RoboDK station: simulation.rdk

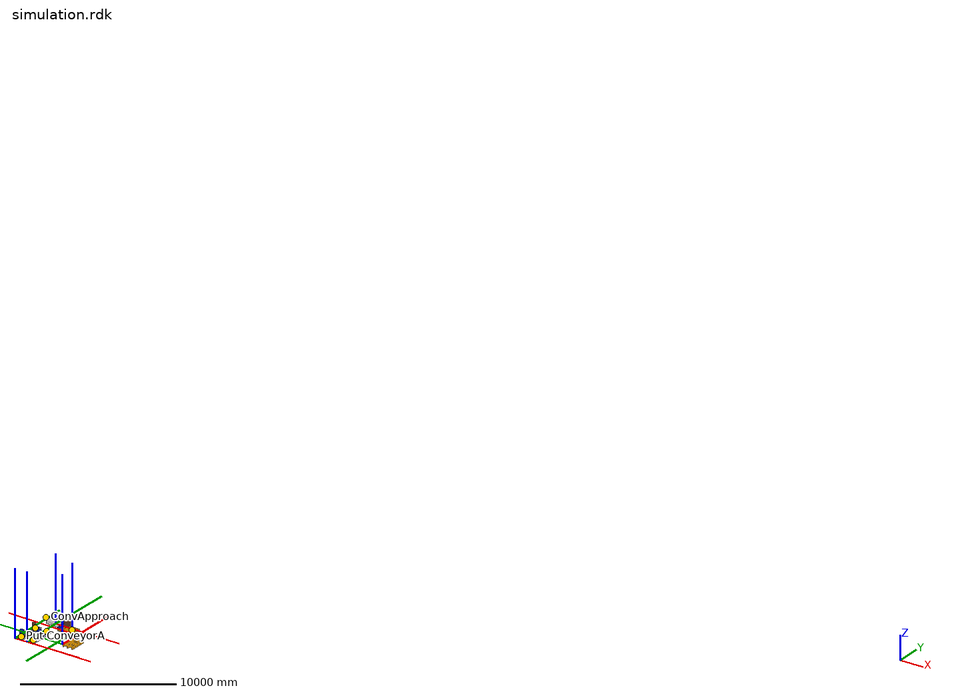
[picture v0: the station drawn from its stored meshes, robots at their saved joint values, targets as dots, program paths as lines]
Station Conveyor simulation. Poses are relative to the parent item; angles as X-Y-Z fixed-axis rotations.
Station parameters (name, value as stored): SizeBox, 150, 300, 150, SizePallet, 3,2,3, ConvSpeed, 40.0, SENSOR, 0, SENSOR-1, 0, SENSOR-2, 0, ROBOT_SWITCHER, 0, TRIGGER-2, 0, TRIGGER-1, 0, SizeBoxA, 240.0,200.0,500.0, SizePalletA, 3,3,3, SizeBoxB, 220.0,190.0,450.0, SizePalletB, 3,3,3, BoxType, 2
  - object box100mm at (0, 0, 0) mm, size 100 x 100 x 100 mm, geometry from box.sld
  - frame ABB IRB 460 Base at (1386.49, 2720.82, 0) mm, rotated rx 0 ry 0 rz -1.04 deg
    - robot ABB IRB 460: 4 axes, payload 110 kg, reach 2400 mm, repeatability 0.2 mm, weight 925 kg
        joint limits [-165, -40, -20, -300] to [165, 85, 120, 300]; home [0, 0, 0, 0]; saved at [-93.5, -29.324, 4.864, 86.5]
      - tool Gripper, TCP at (24.96, -1.82, 200) mm, size 240 x 288 x 203 mm
    - target ConvApproach (joint target) at (-38.73, -1039.73, 855.5) mm, rotated rx -180 ry 0 rz 0 deg; joints [-93.5, -29.324, 4.864, 86.5, 0, 0] of ABB IRB 460
    - target PalletApproach (joint target) at (1357.36, -110.16, 3.72) mm, rotated rx -180 ry 0 rz 0 deg; joints [-4.804, 23.379, 62.26, 175.196, 0, 0] of ABB IRB 460
    - frame PalletB at (545.23, 1038.18, -930) mm, rotated rx 0 ry 0 rz -180 deg
      - object PalletExtension at (1200, -800, 0) mm, rotated rx 0 ry 0 rz 90 deg, size 800 x 144 x 1200 mm, geometry from User Library-Europallet.igs
    - frame Pallet at (973.14, -611.03, -930) mm, rotated rx 0 ry 0 rz 90 deg
      - object Europallet at (1200, -800, 0) mm, rotated rx 0 ry 0 rz 90 deg, size 800 x 144 x 1200 mm, geometry from User Library-Europallet.igs
      - object Part 2 1030.0 685.0 225.0 1.0 at (2351.1, 1457.91, 225) mm, rotated rx -180 ry 0 rz -90 deg, size 220 x 190 x 450 mm, geometry from box.sld
      - object Part 2 1030.0 495.0 225.0 1.0 at (2149.1, 1457.91, 225) mm, rotated rx -180 ry 0 rz -90 deg, size 220 x 190 x 450 mm, geometry from box.sld
      - object Part 1 1080.0 300.0 250.0 1.0 at (1950.1, 1507.91, 250) mm, rotated rx -180 ry 0 rz -90 deg, size 240 x 200 x 500 mm, geometry from box.sld
      - object Part 1 1080.0 100.0 250.0 1.0 at (1779.1, 1507.91, 250) mm, rotated rx -180 ry 0 rz -90 deg, size 240 x 200 x 500 mm, geometry from box.sld
      - object Part 2 810.0 685.0 225.0 1.0 at (2343.1, 1237.91, 225) mm, rotated rx -180 ry 0 rz -90 deg, size 220 x 190 x 450 mm, geometry from box.sld
      - object Part 2 810.0 495.0 225.0 1.0 at (2144.1, 1237.91, 225) mm, rotated rx -180 ry 0 rz -90 deg, size 220 x 190 x 450 mm, geometry from box.sld
  - frame ConveyorReferenceA at (597.23, -679.82, 119.18) mm
    - robot Conveyor BeltA: 1 axes
        modified DH rows (alpha deg, a mm, theta deg, d mm): 0, 0, 0, 0 linear
        base shift (440, 200, 0) mm, rotated rx 0 ry 90 rz 90 deg
        joint limits [-500000] to [500000]; home [0]; saved at [-494037]
      - frame MovingRefA at (0, 0, 0) mm
        - object Part 2 590.0 685.0 225.0 1.0 at (495646.12, 240, 225) mm, rotated rx -180 ry 0 rz 90 deg, size 220 x 190 x 450 mm, geometry from box.sld
        - object Part 1 840.0 100.0 250.0 1.0 at (494259.12, 240, 250) mm, rotated rx -180 ry 0 rz 90 deg, size 240 x 200 x 500 mm, geometry from box.sld
        - object Part 2 590.0 495.0 225.0 1.0 at (494259.12, 240, 225) mm, rotated rx -180 ry 0 rz 90 deg, size 220 x 190 x 450 mm, geometry from box.sld
        - object Part 1 600.0 300.0 250.0 1.0 at (494259.12, 240, 250) mm, rotated rx -180 ry 0 rz 90 deg, size 240 x 200 x 500 mm, geometry from box.sld
        - object Part 1 600.0 100.0 250.0 1.0 at (494259.12, 240, 250) mm, rotated rx -180 ry 0 rz 90 deg, size 240 x 200 x 500 mm, geometry from box.sld
        - object Part 2 370.0 305.0 225.0 1.0 at (494259.12, 240, 225) mm, rotated rx -180 ry 0 rz 90 deg, size 220 x 190 x 450 mm, geometry from box.sld
        - object Part 2 150.0 305.0 225.0 1.0 at (494259.12, 240, 225) mm, rotated rx -180 ry 0 rz 90 deg, size 220 x 190 x 450 mm, geometry from box.sld
        - object Part 2 1030.0 685.0 675.0 2.0 at (494259.12, 240, 225) mm, rotated rx -180 ry 0 rz 90 deg, size 220 x 190 x 450 mm, geometry from box.sld
        - object Part 1 1080.0 300.0 750.0 2.0 at (494259.12, 240, 250) mm, rotated rx -180 ry 0 rz 90 deg, size 240 x 200 x 500 mm, geometry from box.sld
        - object Part 2 810.0 685.0 675.0 2.0 at (494259.12, 240, 225) mm, rotated rx -180 ry 0 rz 90 deg, size 220 x 190 x 450 mm, geometry from box.sld
        - object Part 2 590.0 685.0 675.0 2.0 at (494259.12, 240, 225) mm, rotated rx -180 ry 0 rz 90 deg, size 220 x 190 x 450 mm, geometry from box.sld
        - object Part 1 840.0 100.0 750.0 2.0 at (494259.12, 240, 250) mm, rotated rx -180 ry 0 rz 90 deg, size 240 x 200 x 500 mm, geometry from box.sld
        - object Part 2 590.0 495.0 675.0 2.0 at (494259.12, 240, 225) mm, rotated rx -180 ry 0 rz 90 deg, size 220 x 190 x 450 mm, geometry from box.sld
        - object Part 1 600.0 300.0 750.0 2.0 at (494259.12, 240, 250) mm, rotated rx -180 ry 0 rz 90 deg, size 240 x 200 x 500 mm, geometry from box.sld
        - object Part 1 600.0 100.0 750.0 2.0 at (494259.12, 240, 250) mm, rotated rx -180 ry 0 rz 90 deg, size 240 x 200 x 500 mm, geometry from box.sld
        - object Part 2 370.0 305.0 675.0 2.0 at (494259.12, 240, 225) mm, rotated rx -180 ry 0 rz 90 deg, size 220 x 190 x 450 mm, geometry from box.sld
        - object Part 2 150.0 305.0 675.0 2.0 at (494259.12, 240, 225) mm, rotated rx -180 ry 0 rz 90 deg, size 220 x 190 x 450 mm, geometry from box.sld
        - object Part 2 1030.0 685.0 1125.0 3.0 at (494259.12, 240, 225) mm, rotated rx -180 ry 0 rz 90 deg, size 220 x 190 x 450 mm, geometry from box.sld
        - object Part 1 1080.0 300.0 1250.0 3.0 at (494259.12, 240, 250) mm, rotated rx -180 ry 0 rz 90 deg, size 240 x 200 x 500 mm, geometry from box.sld
        - object Part 2 810.0 685.0 1125.0 3.0 at (494259.12, 240, 225) mm, rotated rx -180 ry 0 rz 90 deg, size 220 x 190 x 450 mm, geometry from box.sld
        - object Part 2 590.0 685.0 1125.0 3.0 at (494259.12, 240, 225) mm, rotated rx -180 ry 0 rz 90 deg, size 220 x 190 x 450 mm, geometry from box.sld
        - object Part 1 840.0 100.0 1250.0 3.0 at (494259.12, 240, 250) mm, rotated rx -180 ry 0 rz 90 deg, size 240 x 200 x 500 mm, geometry from box.sld
        - object Part 2 590.0 495.0 1125.0 3.0 at (494259.12, 240, 225) mm, rotated rx -180 ry 0 rz 90 deg, size 220 x 190 x 450 mm, geometry from box.sld
        - object Part 1 600.0 300.0 1250.0 3.0 at (494259.12, 240, 250) mm, rotated rx -180 ry 0 rz 90 deg, size 240 x 200 x 500 mm, geometry from box.sld
        - object Part 1 600.0 100.0 1250.0 3.0 at (494259.12, 240, 250) mm, rotated rx -180 ry 0 rz 90 deg, size 240 x 200 x 500 mm, geometry from box.sld
        - object Part 2 370.0 305.0 1125.0 3.0 at (494259.12, 240, 225) mm, rotated rx -180 ry 0 rz 90 deg, size 220 x 190 x 450 mm, geometry from box.sld
        - object Part 2 150.0 305.0 1125.0 3.0 at (494259.12, 240, 225) mm, rotated rx -180 ry 0 rz 90 deg, size 220 x 190 x 450 mm, geometry from box.sld
        - object Part 2 1030.0 685.0 1575.0 4.0 at (494259.12, 240, 225) mm, rotated rx -180 ry 0 rz 90 deg, size 220 x 190 x 450 mm, geometry from box.sld
        - object Part 1 1080.0 300.0 1750.0 4.0 at (494259.12, 240, 250) mm, rotated rx -180 ry 0 rz 90 deg, size 240 x 200 x 500 mm, geometry from box.sld
        - object Part 2 810.0 685.0 1575.0 4.0 at (494259.12, 240, 225) mm, rotated rx -180 ry 0 rz 90 deg, size 220 x 190 x 450 mm, geometry from box.sld
        - object Part 2 590.0 685.0 1575.0 4.0 at (494259.12, 240, 225) mm, rotated rx -180 ry 0 rz 90 deg, size 220 x 190 x 450 mm, geometry from box.sld
        - object Part 1 840.0 100.0 1750.0 4.0 at (494259.12, 240, 250) mm, rotated rx -180 ry 0 rz 90 deg, size 240 x 200 x 500 mm, geometry from box.sld
        - object Part 2 590.0 495.0 1575.0 4.0 at (494259.12, 240, 225) mm, rotated rx -180 ry 0 rz 90 deg, size 220 x 190 x 450 mm, geometry from box.sld
        - object Part 1 600.0 300.0 1750.0 4.0 at (494259.12, 240, 250) mm, rotated rx -180 ry 0 rz 90 deg, size 240 x 200 x 500 mm, geometry from box.sld
        - object Part 1 600.0 100.0 1750.0 4.0 at (494259.12, 240, 250) mm, rotated rx -180 ry 0 rz 90 deg, size 240 x 200 x 500 mm, geometry from box.sld
        - object Part 2 370.0 305.0 1575.0 4.0 at (494259.12, 240, 225) mm, rotated rx -180 ry 0 rz 90 deg, size 220 x 190 x 450 mm, geometry from box.sld
        - object Part 2 150.0 305.0 1575.0 4.0 at (494259.12, 240, 225) mm, rotated rx -180 ry 0 rz 90 deg, size 220 x 190 x 450 mm, geometry from box.sld
        - object Part 2 1030.0 685.0 225.0 1.0 at (494259.12, 240, 225) mm, rotated rx -180 ry 0 rz 90 deg, size 220 x 190 x 450 mm, geometry from box.sld
        - object Part 1 1080.0 300.0 250.0 1.0 at (494259.12, 240, 250) mm, rotated rx -180 ry 0 rz 90 deg, size 240 x 200 x 500 mm, geometry from box.sld
        - object Part 2 810.0 685.0 225.0 1.0 at (494259.12, 240, 225) mm, rotated rx -180 ry 0 rz 90 deg, size 220 x 190 x 450 mm, geometry from box.sld
        - object Part 2 590.0 685.0 225.0 1.0 at (494259.12, 240, 225) mm, rotated rx -180 ry 0 rz 90 deg, size 220 x 190 x 450 mm, geometry from box.sld
        - object Part 1 840.0 100.0 250.0 1.0 at (494259.12, 240, 250) mm, rotated rx -180 ry 0 rz 90 deg, size 240 x 200 x 500 mm, geometry from box.sld
        - object Part 2 590.0 495.0 225.0 1.0 at (494259.12, 240, 225) mm, rotated rx -180 ry 0 rz 90 deg, size 220 x 190 x 450 mm, geometry from box.sld
        - object Part 1 600.0 300.0 250.0 1.0 at (494259.12, 240, 250) mm, rotated rx -180 ry 0 rz 90 deg, size 240 x 200 x 500 mm, geometry from box.sld
        - object Part 1 600.0 100.0 250.0 1.0 at (494259.12, 240, 250) mm, rotated rx -180 ry 0 rz 90 deg, size 240 x 200 x 500 mm, geometry from box.sld
        - object Part 2 370.0 305.0 225.0 1.0 at (494259.12, 240, 225) mm, rotated rx -180 ry 0 rz 90 deg, size 220 x 190 x 450 mm, geometry from box.sld
        - object Part 2 150.0 305.0 225.0 1.0 at (494259.12, 240, 225) mm, rotated rx -180 ry 0 rz 90 deg, size 220 x 190 x 450 mm, geometry from box.sld
        - object Part 2 1030.0 685.0 675.0 2.0 at (494259.12, 240, 225) mm, rotated rx -180 ry 0 rz 90 deg, size 220 x 190 x 450 mm, geometry from box.sld
        - object Part 1 1080.0 300.0 750.0 2.0 at (494259.12, 240, 250) mm, rotated rx -180 ry 0 rz 90 deg, size 240 x 200 x 500 mm, geometry from box.sld
        - object Part 2 810.0 685.0 675.0 2.0 at (494259.12, 240, 225) mm, rotated rx -180 ry 0 rz 90 deg, size 220 x 190 x 450 mm, geometry from box.sld
        - object Part 2 590.0 685.0 675.0 2.0 at (494259.12, 240, 225) mm, rotated rx -180 ry 0 rz 90 deg, size 220 x 190 x 450 mm, geometry from box.sld
        - object Part 1 840.0 100.0 750.0 2.0 at (494259.12, 240, 250) mm, rotated rx -180 ry 0 rz 90 deg, size 240 x 200 x 500 mm, geometry from box.sld
        - object Part 2 590.0 495.0 675.0 2.0 at (494259.12, 240, 225) mm, rotated rx -180 ry 0 rz 90 deg, size 220 x 190 x 450 mm, geometry from box.sld
        - object Part 1 600.0 300.0 750.0 2.0 at (494259.12, 240, 250) mm, rotated rx -180 ry 0 rz 90 deg, size 240 x 200 x 500 mm, geometry from box.sld
        - object Part 1 600.0 100.0 750.0 2.0 at (494259.12, 240, 250) mm, rotated rx -180 ry 0 rz 90 deg, size 240 x 200 x 500 mm, geometry from box.sld
        - object Part 2 370.0 305.0 675.0 2.0 at (494259.12, 240, 225) mm, rotated rx -180 ry 0 rz 90 deg, size 220 x 190 x 450 mm, geometry from box.sld
        - object Part 2 150.0 305.0 675.0 2.0 at (494259.12, 240, 225) mm, rotated rx -180 ry 0 rz 90 deg, size 220 x 190 x 450 mm, geometry from box.sld
        - object Part 2 1030.0 685.0 1125.0 3.0 at (494259.12, 240, 225) mm, rotated rx -180 ry 0 rz 90 deg, size 220 x 190 x 450 mm, geometry from box.sld
        - object Part 1 1080.0 300.0 1250.0 3.0 at (494259.12, 240, 250) mm, rotated rx -180 ry 0 rz 90 deg, size 240 x 200 x 500 mm, geometry from box.sld
        - object Part 2 810.0 685.0 1125.0 3.0 at (494259.12, 240, 225) mm, rotated rx -180 ry 0 rz 90 deg, size 220 x 190 x 450 mm, geometry from box.sld
        - object Part 2 590.0 685.0 1125.0 3.0 at (494259.12, 240, 225) mm, rotated rx -180 ry 0 rz 90 deg, size 220 x 190 x 450 mm, geometry from box.sld
        - object Part 1 840.0 100.0 1250.0 3.0 at (494259.12, 240, 250) mm, rotated rx -180 ry 0 rz 90 deg, size 240 x 200 x 500 mm, geometry from box.sld
        - object Part 2 590.0 495.0 1125.0 3.0 at (494259.12, 240, 225) mm, rotated rx -180 ry 0 rz 90 deg, size 220 x 190 x 450 mm, geometry from box.sld
        - object Part 1 600.0 300.0 1250.0 3.0 at (494259.12, 240, 250) mm, rotated rx -180 ry 0 rz 90 deg, size 240 x 200 x 500 mm, geometry from box.sld
        - object Part 1 600.0 100.0 1250.0 3.0 at (494259.12, 240, 250) mm, rotated rx -180 ry 0 rz 90 deg, size 240 x 200 x 500 mm, geometry from box.sld
        - object Part 2 370.0 305.0 1125.0 3.0 at (494259.12, 240, 225) mm, rotated rx -180 ry 0 rz 90 deg, size 220 x 190 x 450 mm, geometry from box.sld
        - object Part 2 150.0 305.0 1125.0 3.0 at (494259.12, 240, 225) mm, rotated rx -180 ry 0 rz 90 deg, size 220 x 190 x 450 mm, geometry from box.sld
        - object Part 2 1030.0 685.0 1575.0 4.0 at (494259.12, 240, 225) mm, rotated rx -180 ry 0 rz 90 deg, size 220 x 190 x 450 mm, geometry from box.sld
        - object Part 1 1080.0 300.0 1750.0 4.0 at (494259.12, 240, 250) mm, rotated rx -180 ry 0 rz 90 deg, size 240 x 200 x 500 mm, geometry from box.sld
        - object Part 2 810.0 685.0 1575.0 4.0 at (494259.12, 240, 225) mm, rotated rx -180 ry 0 rz 90 deg, size 220 x 190 x 450 mm, geometry from box.sld
        - object Part 2 590.0 685.0 1575.0 4.0 at (494259.12, 240, 225) mm, rotated rx -180 ry 0 rz 90 deg, size 220 x 190 x 450 mm, geometry from box.sld
        - object Part 1 840.0 100.0 1750.0 4.0 at (494259.12, 240, 250) mm, rotated rx -180 ry 0 rz 90 deg, size 240 x 200 x 500 mm, geometry from box.sld
        - object Part 2 590.0 495.0 1575.0 4.0 at (494259.12, 240, 225) mm, rotated rx -180 ry 0 rz 90 deg, size 220 x 190 x 450 mm, geometry from box.sld
        - object Part 1 600.0 300.0 1750.0 4.0 at (494259.12, 240, 250) mm, rotated rx -180 ry 0 rz 90 deg, size 240 x 200 x 500 mm, geometry from box.sld
        - object Part 1 600.0 100.0 1750.0 4.0 at (494259.12, 240, 250) mm, rotated rx -180 ry 0 rz 90 deg, size 240 x 200 x 500 mm, geometry from box.sld
        - object Part 2 370.0 305.0 1575.0 4.0 at (494259.12, 240, 225) mm, rotated rx -180 ry 0 rz 90 deg, size 220 x 190 x 450 mm, geometry from box.sld
        - object Part 2 150.0 305.0 1575.0 4.0 at (494259.12, 240, 225) mm, rotated rx -180 ry 0 rz 90 deg, size 220 x 190 x 450 mm, geometry from box.sld
    - target ConveyorHomeA (joint target) at (440, 200, 0) mm, rotated rx 0 ry 0 rz 90 deg; joints [0] of Conveyor BeltA
    - target ConveyorMoveA (joint target) at (440, 99999, 0) mm, rotated rx 0 ry 0 rz 90 deg; joints [99799] of Conveyor BeltA
    - object Sensor SICK WL4S-1 at (551, 1930, 24) mm, rotated rx 90 ry 0 rz 180 deg, size 683.3 x 45.2 x 12.5 mm, geometry from SICK WL4S-3P1330-Order no.1042068 (1).stp
    - target Get ConveyorA (Cartesian target) at (200, 1950, 0) mm, rotated rx -180 ry 0 rz 0 deg; joints [-111.887, 26.233, 48.865, -292.923, 0, 0] of ABB IRB 460
    - target Put ConveyorA (Cartesian target) at (200, 422.12, 0) mm, rotated rx -180 ry 0 rz 180 deg; joints [164.915, -63.548, 110.129, -136.581, -90, -15.085]
  - frame ConveyorReferenceB at (1500, -679.82, 119.18) mm
    - robot Conveyor BeltB: 1 axes
        modified DH rows (alpha deg, a mm, theta deg, d mm): 0, 0, 0, 0 linear
        base shift (440, 200, 0) mm, rotated rx 0 ry 90 rz 90 deg
        joint limits [-500000] to [500000]; home [0]; saved at [-494159]
      - frame MovingRefB at (0, 0, 0) mm
        - object Part 1 840.0 300.0 250.0 1.0 at (495052.11, 240, 250) mm, rotated rx -180 ry 0 rz 90 deg, size 240 x 200 x 500 mm, geometry from box.sld
        - object Part 1 360.0 700.0 250.0 1.0 at (494381.11, 240, 250) mm, rotated rx -180 ry 0 rz 90 deg, size 240 x 200 x 500 mm, geometry from box.sld
        - object Part 1 120.0 700.0 250.0 1.0 at (494381.11, 240, 250) mm, rotated rx -180 ry 0 rz 90 deg, size 240 x 200 x 500 mm, geometry from box.sld
        - object Part 1 360.0 500.0 250.0 1.0 at (494381.11, 240, 250) mm, rotated rx -180 ry 0 rz 90 deg, size 240 x 200 x 500 mm, geometry from box.sld
        - object Part 1 120.0 500.0 250.0 1.0 at (494381.11, 240, 250) mm, rotated rx -180 ry 0 rz 90 deg, size 240 x 200 x 500 mm, geometry from box.sld
        - object Part 2 370.0 115.0 225.0 1.0 at (494381.11, 240, 225) mm, rotated rx -180 ry 0 rz 90 deg, size 220 x 190 x 450 mm, geometry from box.sld
        - object Part 2 150.0 115.0 225.0 1.0 at (494381.11, 240, 225) mm, rotated rx -180 ry 0 rz 90 deg, size 220 x 190 x 450 mm, geometry from box.sld
        - object Part 2 1030.0 495.0 675.0 2.0 at (494381.11, 240, 225) mm, rotated rx -180 ry 0 rz 90 deg, size 220 x 190 x 450 mm, geometry from box.sld
        - object Part 1 1080.0 100.0 750.0 2.0 at (494381.11, 240, 250) mm, rotated rx -180 ry 0 rz 90 deg, size 240 x 200 x 500 mm, geometry from box.sld
        - object Part 2 810.0 495.0 675.0 2.0 at (494381.11, 240, 225) mm, rotated rx -180 ry 0 rz 90 deg, size 220 x 190 x 450 mm, geometry from box.sld
        - object Part 1 840.0 300.0 750.0 2.0 at (494381.11, 240, 250) mm, rotated rx -180 ry 0 rz 90 deg, size 240 x 200 x 500 mm, geometry from box.sld
        - object Part 1 360.0 700.0 750.0 2.0 at (494381.11, 240, 250) mm, rotated rx -180 ry 0 rz 90 deg, size 240 x 200 x 500 mm, geometry from box.sld
        - object Part 1 120.0 700.0 750.0 2.0 at (494381.11, 240, 250) mm, rotated rx -180 ry 0 rz 90 deg, size 240 x 200 x 500 mm, geometry from box.sld
        - object Part 1 360.0 500.0 750.0 2.0 at (494381.11, 240, 250) mm, rotated rx -180 ry 0 rz 90 deg, size 240 x 200 x 500 mm, geometry from box.sld
        - object Part 1 120.0 500.0 750.0 2.0 at (494381.11, 240, 250) mm, rotated rx -180 ry 0 rz 90 deg, size 240 x 200 x 500 mm, geometry from box.sld
        - object Part 2 370.0 115.0 675.0 2.0 at (494381.11, 240, 225) mm, rotated rx -180 ry 0 rz 90 deg, size 220 x 190 x 450 mm, geometry from box.sld
        - object Part 2 150.0 115.0 675.0 2.0 at (494381.11, 240, 225) mm, rotated rx -180 ry 0 rz 90 deg, size 220 x 190 x 450 mm, geometry from box.sld
        - object Part 2 1030.0 495.0 1125.0 3.0 at (494381.11, 240, 225) mm, rotated rx -180 ry 0 rz 90 deg, size 220 x 190 x 450 mm, geometry from box.sld
        - object Part 1 1080.0 100.0 1250.0 3.0 at (494381.11, 240, 250) mm, rotated rx -180 ry 0 rz 90 deg, size 240 x 200 x 500 mm, geometry from box.sld
        - object Part 2 810.0 495.0 1125.0 3.0 at (494381.11, 240, 225) mm, rotated rx -180 ry 0 rz 90 deg, size 220 x 190 x 450 mm, geometry from box.sld
        - object Part 1 840.0 300.0 1250.0 3.0 at (494381.11, 240, 250) mm, rotated rx -180 ry 0 rz 90 deg, size 240 x 200 x 500 mm, geometry from box.sld
        - object Part 1 360.0 700.0 1250.0 3.0 at (494381.11, 240, 250) mm, rotated rx -180 ry 0 rz 90 deg, size 240 x 200 x 500 mm, geometry from box.sld
        - object Part 1 120.0 700.0 1250.0 3.0 at (494381.11, 240, 250) mm, rotated rx -180 ry 0 rz 90 deg, size 240 x 200 x 500 mm, geometry from box.sld
        - object Part 1 360.0 500.0 1250.0 3.0 at (494381.11, 240, 250) mm, rotated rx -180 ry 0 rz 90 deg, size 240 x 200 x 500 mm, geometry from box.sld
        - object Part 1 120.0 500.0 1250.0 3.0 at (494381.11, 240, 250) mm, rotated rx -180 ry 0 rz 90 deg, size 240 x 200 x 500 mm, geometry from box.sld
        - object Part 2 370.0 115.0 1125.0 3.0 at (494381.11, 240, 225) mm, rotated rx -180 ry 0 rz 90 deg, size 220 x 190 x 450 mm, geometry from box.sld
        - object Part 2 150.0 115.0 1125.0 3.0 at (494381.11, 240, 225) mm, rotated rx -180 ry 0 rz 90 deg, size 220 x 190 x 450 mm, geometry from box.sld
        - object Part 2 1030.0 495.0 1575.0 4.0 at (494381.11, 240, 225) mm, rotated rx -180 ry 0 rz 90 deg, size 220 x 190 x 450 mm, geometry from box.sld
        - object Part 1 1080.0 100.0 1750.0 4.0 at (494381.11, 240, 250) mm, rotated rx -180 ry 0 rz 90 deg, size 240 x 200 x 500 mm, geometry from box.sld
        - object Part 2 810.0 495.0 1575.0 4.0 at (494381.11, 240, 225) mm, rotated rx -180 ry 0 rz 90 deg, size 220 x 190 x 450 mm, geometry from box.sld
        - object Part 1 840.0 300.0 1750.0 4.0 at (494381.11, 240, 250) mm, rotated rx -180 ry 0 rz 90 deg, size 240 x 200 x 500 mm, geometry from box.sld
        - object Part 1 360.0 700.0 1750.0 4.0 at (494381.11, 240, 250) mm, rotated rx -180 ry 0 rz 90 deg, size 240 x 200 x 500 mm, geometry from box.sld
        - object Part 1 120.0 700.0 1750.0 4.0 at (494381.11, 240, 250) mm, rotated rx -180 ry 0 rz 90 deg, size 240 x 200 x 500 mm, geometry from box.sld
        - object Part 1 360.0 500.0 1750.0 4.0 at (494381.11, 240, 250) mm, rotated rx -180 ry 0 rz 90 deg, size 240 x 200 x 500 mm, geometry from box.sld
        - object Part 1 120.0 500.0 1750.0 4.0 at (494381.11, 240, 250) mm, rotated rx -180 ry 0 rz 90 deg, size 240 x 200 x 500 mm, geometry from box.sld
        - object Part 2 370.0 115.0 1575.0 4.0 at (494381.11, 240, 225) mm, rotated rx -180 ry 0 rz 90 deg, size 220 x 190 x 450 mm, geometry from box.sld
        - object Part 2 150.0 115.0 1575.0 4.0 at (494381.11, 240, 225) mm, rotated rx -180 ry 0 rz 90 deg, size 220 x 190 x 450 mm, geometry from box.sld
        - object Part 2 1030.0 495.0 225.0 1.0 at (494381.11, 240, 225) mm, rotated rx -180 ry 0 rz 90 deg, size 220 x 190 x 450 mm, geometry from box.sld
        - object Part 1 1080.0 100.0 250.0 1.0 at (494381.11, 240, 250) mm, rotated rx -180 ry 0 rz 90 deg, size 240 x 200 x 500 mm, geometry from box.sld
        - object Part 2 810.0 495.0 225.0 1.0 at (494381.11, 240, 225) mm, rotated rx -180 ry 0 rz 90 deg, size 220 x 190 x 450 mm, geometry from box.sld
        - object Part 1 840.0 300.0 250.0 1.0 at (494381.11, 240, 250) mm, rotated rx -180 ry 0 rz 90 deg, size 240 x 200 x 500 mm, geometry from box.sld
        - object Part 1 360.0 700.0 250.0 1.0 at (494381.11, 240, 250) mm, rotated rx -180 ry 0 rz 90 deg, size 240 x 200 x 500 mm, geometry from box.sld
        - object Part 1 120.0 700.0 250.0 1.0 at (494381.11, 240, 250) mm, rotated rx -180 ry 0 rz 90 deg, size 240 x 200 x 500 mm, geometry from box.sld
        - object Part 1 360.0 500.0 250.0 1.0 at (494381.11, 240, 250) mm, rotated rx -180 ry 0 rz 90 deg, size 240 x 200 x 500 mm, geometry from box.sld
        - object Part 1 120.0 500.0 250.0 1.0 at (494381.11, 240, 250) mm, rotated rx -180 ry 0 rz 90 deg, size 240 x 200 x 500 mm, geometry from box.sld
        - object Part 2 370.0 115.0 225.0 1.0 at (494381.11, 240, 225) mm, rotated rx -180 ry 0 rz 90 deg, size 220 x 190 x 450 mm, geometry from box.sld
        - object Part 2 150.0 115.0 225.0 1.0 at (494381.11, 240, 225) mm, rotated rx -180 ry 0 rz 90 deg, size 220 x 190 x 450 mm, geometry from box.sld
        - object Part 2 1030.0 495.0 675.0 2.0 at (494381.11, 240, 225) mm, rotated rx -180 ry 0 rz 90 deg, size 220 x 190 x 450 mm, geometry from box.sld
        - object Part 1 1080.0 100.0 750.0 2.0 at (494381.11, 240, 250) mm, rotated rx -180 ry 0 rz 90 deg, size 240 x 200 x 500 mm, geometry from box.sld
        - object Part 2 810.0 495.0 675.0 2.0 at (494381.11, 240, 225) mm, rotated rx -180 ry 0 rz 90 deg, size 220 x 190 x 450 mm, geometry from box.sld
        - object Part 1 840.0 300.0 750.0 2.0 at (494381.11, 240, 250) mm, rotated rx -180 ry 0 rz 90 deg, size 240 x 200 x 500 mm, geometry from box.sld
        - object Part 1 360.0 700.0 750.0 2.0 at (494381.11, 240, 250) mm, rotated rx -180 ry 0 rz 90 deg, size 240 x 200 x 500 mm, geometry from box.sld
        - object Part 1 120.0 700.0 750.0 2.0 at (494381.11, 240, 250) mm, rotated rx -180 ry 0 rz 90 deg, size 240 x 200 x 500 mm, geometry from box.sld
        - object Part 1 360.0 500.0 750.0 2.0 at (494381.11, 240, 250) mm, rotated rx -180 ry 0 rz 90 deg, size 240 x 200 x 500 mm, geometry from box.sld
        - object Part 1 120.0 500.0 750.0 2.0 at (494381.11, 240, 250) mm, rotated rx -180 ry 0 rz 90 deg, size 240 x 200 x 500 mm, geometry from box.sld
        - object Part 2 370.0 115.0 675.0 2.0 at (494381.11, 240, 225) mm, rotated rx -180 ry 0 rz 90 deg, size 220 x 190 x 450 mm, geometry from box.sld
        - object Part 2 150.0 115.0 675.0 2.0 at (494381.11, 240, 225) mm, rotated rx -180 ry 0 rz 90 deg, size 220 x 190 x 450 mm, geometry from box.sld
        - object Part 2 1030.0 495.0 1125.0 3.0 at (494381.11, 240, 225) mm, rotated rx -180 ry 0 rz 90 deg, size 220 x 190 x 450 mm, geometry from box.sld
        - object Part 1 1080.0 100.0 1250.0 3.0 at (494381.11, 240, 250) mm, rotated rx -180 ry 0 rz 90 deg, size 240 x 200 x 500 mm, geometry from box.sld
        - object Part 2 810.0 495.0 1125.0 3.0 at (494381.11, 240, 225) mm, rotated rx -180 ry 0 rz 90 deg, size 220 x 190 x 450 mm, geometry from box.sld
        - object Part 1 840.0 300.0 1250.0 3.0 at (494381.11, 240, 250) mm, rotated rx -180 ry 0 rz 90 deg, size 240 x 200 x 500 mm, geometry from box.sld
        - object Part 1 360.0 700.0 1250.0 3.0 at (494381.11, 240, 250) mm, rotated rx -180 ry 0 rz 90 deg, size 240 x 200 x 500 mm, geometry from box.sld
        - object Part 1 120.0 700.0 1250.0 3.0 at (494381.11, 240, 250) mm, rotated rx -180 ry 0 rz 90 deg, size 240 x 200 x 500 mm, geometry from box.sld
        - object Part 1 360.0 500.0 1250.0 3.0 at (494381.11, 240, 250) mm, rotated rx -180 ry 0 rz 90 deg, size 240 x 200 x 500 mm, geometry from box.sld
        - object Part 1 120.0 500.0 1250.0 3.0 at (494381.11, 240, 250) mm, rotated rx -180 ry 0 rz 90 deg, size 240 x 200 x 500 mm, geometry from box.sld
        - object Part 2 370.0 115.0 1125.0 3.0 at (494381.11, 240, 225) mm, rotated rx -180 ry 0 rz 90 deg, size 220 x 190 x 450 mm, geometry from box.sld
        - object Part 2 150.0 115.0 1125.0 3.0 at (494381.11, 240, 225) mm, rotated rx -180 ry 0 rz 90 deg, size 220 x 190 x 450 mm, geometry from box.sld
        - object Part 2 1030.0 495.0 1575.0 4.0 at (494381.11, 240, 225) mm, rotated rx -180 ry 0 rz 90 deg, size 220 x 190 x 450 mm, geometry from box.sld
        - object Part 1 1080.0 100.0 1750.0 4.0 at (494381.11, 240, 250) mm, rotated rx -180 ry 0 rz 90 deg, size 240 x 200 x 500 mm, geometry from box.sld
        - object Part 2 810.0 495.0 1575.0 4.0 at (494381.11, 240, 225) mm, rotated rx -180 ry 0 rz 90 deg, size 220 x 190 x 450 mm, geometry from box.sld
        - object Part 1 840.0 300.0 1750.0 4.0 at (494381.11, 240, 250) mm, rotated rx -180 ry 0 rz 90 deg, size 240 x 200 x 500 mm, geometry from box.sld
        - object Part 1 360.0 700.0 1750.0 4.0 at (494381.11, 240, 250) mm, rotated rx -180 ry 0 rz 90 deg, size 240 x 200 x 500 mm, geometry from box.sld
        - object Part 1 120.0 700.0 1750.0 4.0 at (494381.11, 240, 250) mm, rotated rx -180 ry 0 rz 90 deg, size 240 x 200 x 500 mm, geometry from box.sld
        - object Part 1 360.0 500.0 1750.0 4.0 at (494381.11, 240, 250) mm, rotated rx -180 ry 0 rz 90 deg, size 240 x 200 x 500 mm, geometry from box.sld
        - object Part 1 120.0 500.0 1750.0 4.0 at (494381.11, 240, 250) mm, rotated rx -180 ry 0 rz 90 deg, size 240 x 200 x 500 mm, geometry from box.sld
        - object Part 2 370.0 115.0 1575.0 4.0 at (494381.11, 240, 225) mm, rotated rx -180 ry 0 rz 90 deg, size 220 x 190 x 450 mm, geometry from box.sld
        - object Part 2 150.0 115.0 1575.0 4.0 at (494381.11, 240, 225) mm, rotated rx -180 ry 0 rz 90 deg, size 220 x 190 x 450 mm, geometry from box.sld
    - target ConveyorHomeB (joint target) at (440, 200, 0) mm, rotated rx 0 ry 0 rz 90 deg; joints [0] of Conveyor BeltB
    - target ConveyorMoveB (joint target) at (440, 99999, 0) mm, rotated rx 0 ry 0 rz 90 deg; joints [99799, 0, 0, 0, 0, 0] of Conveyor BeltB
    - object Sensor SICK WL4S-2 at (551, 1930, 24) mm, rotated rx 90 ry 0 rz 180 deg, size 683.3 x 45.2 x 12.5 mm, geometry from SICK WL4S-3P1330-Order no.1042068 (1).stp
    - target Get ConveyorB (Cartesian target) at (200, 1950, 0) mm, rotated rx -180 ry 0 rz 0 deg; joints [-77.728, 22.073, 51.31, -258.764, 0, 0] of ABB IRB 460
    - target Put ConveyorB (Cartesian target) at (200, 422.12, 0) mm, rotated rx -180 ry 0 rz 180 deg; joints [164.915, -63.548, 110.129, -136.581, -90, -15.085]
  - Python program SetSimulationParams (listed below)
  - Python program AddBox (listed below)
  - Python program SensorActivate_1 (listed below)
  - Python program SensorActivate_2 (listed below)
  - Python program RobotC_StoreParts (listed below)
  - program MoveConveyorA (1 instructions, listed below)
  - program MoveConveyorB (1 instructions, listed below)
  - program MainSimulation (6 instructions, listed below)

--- Python program SetSimulationParams ---
# Type help("robolink") or help("robodk") for more information
# Press F5 to run the script
# Note: you do not need to keep a copy of this file, your python script is saved with the station
from robolink import *    # API to communicate with RoboDK
from robodk import *      # basic matrix operations


RDK = Robolink()


PARAM_SIZE_BOX_A = 'SizeBoxA'
size_box_A = RDK.getParam(PARAM_SIZE_BOX_A)

# ------------------------------------------------------------
size_box_input_A = mbox('Box size PALLET A in mm | FORMAT: L,W,H', entry=size_box_A)
if size_box_input_A:
    RDK.setParam(PARAM_SIZE_BOX_A, size_box_input_A)
else:
    raise Exception('Operation cancelled by user')



PARAM_SIZE_BOX_B = 'SizeBoxB'
size_box_B = RDK.getParam(PARAM_SIZE_BOX_B)

# ------------------------------------------------------------
size_box_input_B = mbox('Box size PALLET B in mm | FORMAT: L,W,H', entry=size_box_B)
if size_box_input_B:
    RDK.setParam(PARAM_SIZE_BOX_B, size_box_input_B)
else:
    raise Exception('Operation cancelled by user')

--- Python program AddBox ---
# Type help("robolink") or help("robodk") for more information
# Press F5 to run the script
# Note: you do not need to keep a copy of this file, your python script is saved with the station
from robolink import *    # API to communicate with RoboDK
from robodk import *      # basic matrix operations
import random
RDK = Robolink()

PART_NAME = 'box100mm'

def cleanup(objects, startswith="Part "):
    """Deletes all objects where the name starts with "startswith", from the provided list of objects."""
    for item in objects:
        if item.Name().startswith(startswith):
            item.Delete()

all_objects = RDK.ItemList(ITEM_TYPE_OBJECT, False)
cleanup(all_objects, 'Part')
all_tools = RDK.ItemList(ITEM_TYPE_TOOL, False)
cleanup(all_tools, 'TCP ')



def get_row_data(row):
    data = []
    row += " "
    aux = ""

    for i in range(len(row)):
        if (row[i].isalpha() or row[i].isdigit() or row[i] == '.' or row[i] == '(' or row[i] == ')' or row[i] == '°' and row[i] != " "):
            aux += row[i]
        else:
            if len(aux) > 1:
                data.append(aux)
                aux = ""

    data[0] = data[0].split('(')[0]

    return data

part_data = []

try:
    f = open("Pattern.txt", "r")
    for x in f:
        data = get_row_data(x)
        useful_data = data[0] + " " + data[1] + " " + data[2] + " " + data[3] + " " + data[7]
        part_data.append(useful_data)
    f.close()

except:
    mbox("Could not read the file: make sure the file is named: Pattern.txt and it is in the right place")


#read from file the sizes
boxes_number = len(part_data)

#time between boxes
pause_time = 5.5

SIZE_BOX_A = RDK.getParam('SizeBoxA')
SIZE_BOX_B = RDK.getParam('SizeBoxB')

target_conv_a = RDK.Item('Put ConveyorA', ITEM_TYPE_TARGET)
target_conv_b = RDK.Item('Put ConveyorB', ITEM_TYPE_TARGET)

SIZE_BOX_XYZ_A = [float(x.replace(' ','')) for x in SIZE_BOX_A.split(',')]
SIZE_BOX_XYZ_B = [float(x.replace(' ','')) for x in SIZE_BOX_B.split(',')]

part_item = RDK.Item(PART_NAME, ITEM_TYPE_OBJECT)

conveyor_ref_A = RDK.Item('MovingRefA', ITEM_TYPE_FRAME)
conveyor_ref_B = RDK.Item('MovingRefB', ITEM_TYPE_FRAME)


for i in range(2):
    n = 0
    while n < boxes_number:

        conveyor_ref = None
        target_conv = None
        SIZE_BOX = None
        SIZE_BOX_XYZ = None

        box_type = part_data[n][0]

        if (box_type == "1"):
            SIZE_BOX = SIZE_BOX_A
            SIZE_BOX_XYZ = SIZE_BOX_XYZ_A

        if (box_type == "2"):
            SIZE_BOX = SIZE_BOX_B
            SIZE_BOX_XYZ = SIZE_BOX_XYZ_B

        if (n % 2 == 0):
            conveyor_ref = conveyor_ref_A
            target_conv = target_conv_a

        if (n % 2 == 1):
            conveyor_ref = conveyor_ref_B
            target_conv = target_conv_b

        [SIZE_BOX_X, SIZE_BOX_Y, SIZE_BOX_Z] = SIZE_BOX_XYZ

        # Create a new part and place it on top of the conveyor, adjusting the height
        part_pos = target_conv.PoseAbs() * transl(0,0, -SIZE_BOX_Z)
        part_item.Copy()
        newpart = conveyor_ref.Paste()
        newpart.setPoseAbs(part_pos*transl(0,0,SIZE_BOX_Z/2))
        newpart.setName('Part ' + part_data[n])
        #newpart.setName('Part 2 1075.0 720.0 1750.0 1')
        newpart.Scale([SIZE_BOX_X/100, SIZE_BOX_Y/100, SIZE_BOX_Z/100]) #scale with respect to the reference object (100mm cube)
        newpart.setVisible(True, False) #make item visible but hide the reference frame


        if (part_data[n][0] == '1'):
            newpart.Recolor([0.1, 0.2, 0.8, 1])  # set RGBA color
        else:
            newpart.Recolor([0.5, 0.3, 0.2, 1])  # set RGBA color
        n = n + 1

        pause(pause_time)

--- Python program SensorActivate_1 ---
# Type help("robolink") or help("robodk") for more information
# Press F5 to run the script
# Note: you do not need to keep a copy of this file, your python script is saved with the station
from robolink import *    # API to communicate with RoboDK
from robodk import *      # basic matrix operations
RDK = Robolink()

# This script allows to simulate a laser sensor
# that detect the presence of a part in a plane,
# such as a part crossing a laser sensor in a
# conveyor belt

# Use a target from the station as a reference plane:
SENSOR_NAME = 'Sensor SICK WL4S-1'
SENSOR_VARIABLE = 'SENSOR-1'

# Look for parts with the keyword "Part"
PART_KEYWORD = 'Part '

# Update status every 1 ms
RECHECK_PERIOD = 0.01

# Get the sensor and the detection plane
SENSOR = RDK.Item(SENSOR_NAME, ITEM_TYPE_OBJECT)

pause(2.0)

OBJECTS_REFERENCE = 'MovingRefA'
moving_ref = RDK.Item(OBJECTS_REFERENCE, ITEM_TYPE_FRAME)

# Loop forever to detect parts
detected_status = -1

pause_time = 3

while True:
    detected = 0
    for obj in moving_ref.Childs():
        # check if an object has the part keyword and is detected by the laser
        if SENSOR.Collision(obj) > 0:
            try:
                data = obj.Name().split(' ')
                RDK.setParam('BoxType', int(data[1]))
                #size_box_input = mbox('COLL')
                detected = 1
            except:
                pass
            break

    # update the current status of the sensor
    if detected_status != detected:
        detected_status = detected
        RDK.setParam(SENSOR_VARIABLE, detected_status)
        pause(pause_time - 1)

    # Wait some time...
    pause(RECHECK_PERIOD)

--- Python program SensorActivate_2 ---
# Type help("robolink") or help("robodk") for more information
# Press F5 to run the script
# Note: you do not need to keep a copy of this file, your python script is saved with the station
from robolink import *    # API to communicate with RoboDK
from robodk import *      # basic matrix operations
RDK = Robolink()

# This script allows to simulate a laser sensor
# that detect the presence of a part in a plane,
# such as a part crossing a laser sensor in a
# conveyor belt

# Use a target from the station as a reference plane:
SENSOR_NAME = 'Sensor SICK WL4S-2'
SENSOR_VARIABLE = 'SENSOR-2'

# Look for parts with the keyword "Part"
PART_KEYWORD = 'Part '

# Update status every 1 ms
RECHECK_PERIOD = 0.01

# Get the sensor and the detection plane
SENSOR = RDK.Item(SENSOR_NAME, ITEM_TYPE_OBJECT)

pause(2.0)

OBJECTS_REFERENCE = 'MovingRefB'
moving_ref = RDK.Item(OBJECTS_REFERENCE, ITEM_TYPE_FRAME)

pause_time = 3

# Loop forever to detect parts
detected_status = -1
while True:
    detected = 0

    for obj in moving_ref.Childs():
        # check if an object has the part keyword and is detected by the laser
        if SENSOR.Collision(obj) > 0:
            try:
                data = obj.Name().split(' ')
                RDK.setParam('BoxType', int(data[1]))
                #size_box_input = mbox('COLL')
                detected = 1
            except:
                pass
            break

    # update the current status of the sensor
    if detected_status != detected:
        detected_status = detected
        RDK.setParam(SENSOR_VARIABLE, detected_status)
        pause(pause_time - 1)

    # Wait some time...
    pause(RECHECK_PERIOD)

--- Python program RobotC_StoreParts ---
# Type help("robolink") or help("robodk") for more information
# Press F5 to run the script
# Note: you do not need to keep a copy of this file, your python script is saved with the station
from robolink import *    # API to communicate with RoboDK
from robodk import *      # basic matrix operations
from random import uniform

# Use RoboDK API as RL
RDK = Robolink()

# define default approach distance
APPROACH = 0

# gather robot, tool and reference frames from the station
robot               = RDK.Item('ABB IRB 460', ITEM_TYPE_ROBOT)
tool                = RDK.Item('Gripper', ITEM_TYPE_TOOL)

# gather targets
target_pallet_safe = RDK.Item('PalletApproach', ITEM_TYPE_TARGET)
target_conv_safe = RDK.Item('ConvApproach', ITEM_TYPE_TARGET)

# get variable parameters
SIZE_BOX_A = RDK.getParam('SizeBoxA')
SIZE_BOX_XYZ_A = [float(x.replace(' ','')) for x in SIZE_BOX_A.split(',')]
SIZE_BOX_Z_A = SIZE_BOX_XYZ_A[2] # the height of the boxes is important to take into account when approaching the positions

SIZE_BOX_B = RDK.getParam('SizeBoxB')
SIZE_BOX_XYZ_B = [float(x.replace(' ','')) for x in SIZE_BOX_B.split(',')]
SIZE_BOX_Z_B = SIZE_BOX_XYZ_B[2] # the height of the boxes is important to take into account when approaching the positions

def TCP_On(toolitem):
    """Attaches the closest object to the toolitem Htool pose,
    It will also output appropriate function calls on the generated robot program (call to TCP_On)"""
    toolitem.AttachClosest()
    toolitem.RDK().RunMessage('Set air valve on')
    toolitem.RDK().RunProgram('TCP_On()');

def TCP_Off(toolitem, itemleave=0):
    """Detaches the closest object attached to the toolitem Htool pose,
    It will also output appropriate function calls on the generated robot program (call to TCP_Off)"""
    #toolitem.DetachClosest(itemleave)
    toolitem.DetachAll(itemleave)
    toolitem.RDK().RunMessage('Set air valve off')
    toolitem.RDK().RunProgram('TCP_Off()');

def cleanup(objects, startswith="Part "):
    """Deletes all objects where the name starts with "startswith", from the provided list of objects."""
    for item in objects:
        if item.Name().startswith(startswith):
            item.Delete()



# Calculate a new TCP that takes into account the size of the part (targets are set to the center of the box)


# ---------------------------------------------------------------------------------
# -------------------------- PROGRAM START ----------------------------------------

RDK.setParam('SENSOR-1', 0)
RDK.setParam('SENSOR-2', 0)


file_data_rows = 0
for line in open("Pattern.txt"): file_data_rows += 1

frame_pallet_b = RDK.Item('PalletB', ITEM_TYPE_FRAME)
frame_pallet = RDK.Item('Pallet', ITEM_TYPE_FRAME)

i = 0
while True:

    #approach conv area
    robot.MoveJ(target_conv_safe)

    target_conv = None
    frame_conv  = None
    SIZE_BOX_Z = None

    all_tools = RDK.ItemList(ITEM_TYPE_TOOL, False)
    cleanup(all_tools, 'TCP ')

    while RDK.getParam('SENSOR-1') == 0 and RDK.getParam('SENSOR-2') == 0:
        pause(0.001)

    if RDK.getParam('SENSOR-1') == 1:
        target_conv = RDK.Item('Get ConveyorA', ITEM_TYPE_TARGET)
        frame_conv  = RDK.Item('ConveyorReferenceA', ITEM_TYPE_FRAME)


    if RDK.getParam('SENSOR-2') == 1:
        target_conv = RDK.Item('Get ConveyorB', ITEM_TYPE_TARGET)
        frame_conv  = RDK.Item('ConveyorReferenceB', ITEM_TYPE_FRAME)


    if RDK.getParam('BoxType') == 1:
        SIZE_BOX_Z = SIZE_BOX_Z_A
        tool_xyzrpw = tool.PoseTool() * transl(0, 0, SIZE_BOX_Z / 2)
        tool_tcp = robot.AddTool(tool_xyzrpw, 'TCP C')
        robot.setPoseTool(tool_tcp)

    if RDK.getParam('BoxType') == 2:
        SIZE_BOX_Z = SIZE_BOX_Z_B
        tool_xyzrpw = tool.PoseTool() * transl(0, 0, SIZE_BOX_Z / 2)
        tool_tcp = robot.AddTool(tool_xyzrpw, 'TCP C')
        robot.setPoseTool(tool_tcp)

    # approach to the conveyor
    robot.setPoseFrame(frame_conv)

    #box position to be picked considering the conveyor frame
    target_conv_pose = target_conv.Pose()*transl(0,0,-SIZE_BOX_Z/2)

    #how to approach the conveyor band
    target_conv_app = target_conv_pose*transl(0,0,-APPROACH)


    #then approach the conveyour
    robot.MoveJ(target_conv_app)


    #go get the box
    robot.MoveL(target_conv_pose)
    TCP_On(tool)

    #safely exit the conveyor frame
    robot.MoveL(target_conv_app)

    #go to the safe point
    robot.MoveJ(target_conv_safe)




 	#--------------------------------------------

    if i < file_data_rows:
        robot.setPoseFrame(frame_pallet_b)
    else:
        robot.setPoseFrame(frame_pallet)

    #BOX DETAILS
    pos_x = 0
    pos_y = 0
    pos_z = 0

    #get the box name to get the info
    box_name = ""
    for box in tool.Childs():
        #mbox(box.Name())
        data = box.Name().split(' ')
        pos_x = float(data[2])
        pos_y = float(data[3])
        pos_z = float(data[4])
        box_name = box.Name()

    #mbox(str([pos_x, pos_y, pos_z]))
    part_position_i = [pos_x, -pos_y, pos_z]

    target_i = transl(part_position_i) * rotx(pi)
    target_i_app = target_i * transl(0,0,-(SIZE_BOX_Z/2))

    robot.MoveJ(target_i_app)

    #place the box
    robot.MoveL(target_i)
    TCP_Off(tool, frame_pallet) # attach the closest part

    robot.MoveJ(target_i_app)

    i = i + 1

--- program MoveConveyorA (robot Conveyor BeltA) ---
  MoveJ (ConveyorMoveA)

--- program MoveConveyorB (robot Conveyor BeltB) ---
  MoveJ (ConveyorMoveB)

--- program MainSimulation ---
  Run MoveConveyorA
  Run MoveConveyorB
  Run SensorActivate_1
  Run SensorActivate_2
  Run AddBox
  Call RobotC_StoreParts
